FUNCTION_BLOCK CompositeBlockWithoutConnections
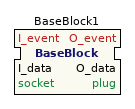
  FBS
    BaseBlock1 : BaseBlock;
  END_FBS
END_FUNCTION_BLOCK
